TYPE XyTableComRequest :
STRUCT
  Start : BOOL;
  Stop : BOOL;
  GoHome : BOOL;
  Halt : BOOL;
END_STRUCT
END_TYPE

(* stored: Version 1.1.0.1
   DUT XyTableComRequest: Id {03a8839c-76f6-47d1-a31e-a1c71504839d} *)
